Fanuc KAREL source: kf00117.KL

PROGRAM KF00117
%NOLOCKGROUP
VAR
I:INTEGER;J:INTEGER;X:REAL;Y:REAL;B:BOOLEAN;C:BOOLEAN;TXT : STRING[80];TXT2 : STRING[80];AI : ARRAY[4] OF INTEGER;BI : ARRAY[4] OF INTEGER;P : XYZWPR
JP : JOINTPOS9
PF : POSITION
V1 : VECTOR
V2 : VECTOR
STATUS:INTEGER
ROUTINE PASSARR(P1:ARRAY[*] OF INTEGER)
BEGIN
--
--
--
--
--
--
--
--
--
--
I=P1[1]
END PASSARR
BEGIN
PASSARR(AI)
END KF00117
